// TwinCAT 3 PLC project Carro_Basico_PLC
// ProgramVersion: 3.1.4024.0
// libraries:
//   Tc2_Standard, * (Beckhoff Automation GmbH)
//   Tc2_System, * (Beckhoff Automation GmbH)
//   Tc3_Module, * (Beckhoff Automation GmbH)
//   VisuDialogs, * (System)
// project tree:
//   / GlobalTextList.TcGTLO, PlcTask.TcTTO, Visualization Manager.TcVMO (not stored)
//   POUs/ FB_Blink.TcPOU (not stored), FB_Carro_DRC_LD.TcPOU, FB_Carro_GRF_LD_M.TcPOU (not stored), FB_Carro_GRF_SFC.TcPOU, FB_Carro_GRF_ST.TcPOU, MAIN.TcPOU
//   VISUs/ V_Carro.TcVIS
// real-time tasks:
//   TASK PlcTask: cycle T#10ms, priority 20, ADS port 350

CONFIGURATION Carro_Basico_PLC
    RESOURCE PLC ON TwinCAT3
        TASK PlcTask(INTERVAL := T#10ms, PRIORITY := 20);
        PROGRAM MAIN WITH PlcTask : MAIN;
    END_RESOURCE
END_CONFIGURATION

// ---- POUs/MAIN.TcPOU
PROGRAM MAIN
VAR
    // Carro: FB_Carro_DRC_LD;
    // Carro: FB_Carro_GRF_SFC;
    // Carro: FB_Carro_GRF_ST;
    Carro: FB_Carro_GRF_LD_M;
END_VAR

Carro();

END_PROGRAM

// ---- POUs/FB_Carro_DRC_LD.TcPOU
FUNCTION_BLOCK FB_Carro_DRC_LD
VAR_INPUT
    ManiobrasTotales: UINT := 2;
    TiempoEspera: TIME := T#2S;
END_VAR
VAR_OUTPUT
    ManiobrasPendientes: UINT;
    TiempoPendiente: TIME;
END_VAR
VAR
    // Estados futuros
    MarchaDerechaFuturo: BOOL;
    MarchaIzquierdaFuturo: BOOL;
    
    // Bloques funcionales
    FlancoPulsadorMarcha: R_TRIG;
    Intermitencia: FB_Blink;
    TemporizadorEspera: TON;
    ContadorManiobras: CTD;
    
    // Entradas
    i_PulsadorMarcha AT %I*: BOOL;
    i_FinalCarreraIzquierda AT %I*: BOOL := TRUE;
    i_FinalCarreraDerecha AT %I*: BOOL;
    
    // Salidas
    o_MarchaIzquierda AT %I*: BOOL;
    o_MarchaDerecha AT %I*: BOOL;
    o_LamparaMarcha AT %I*: BOOL;
END_VAR

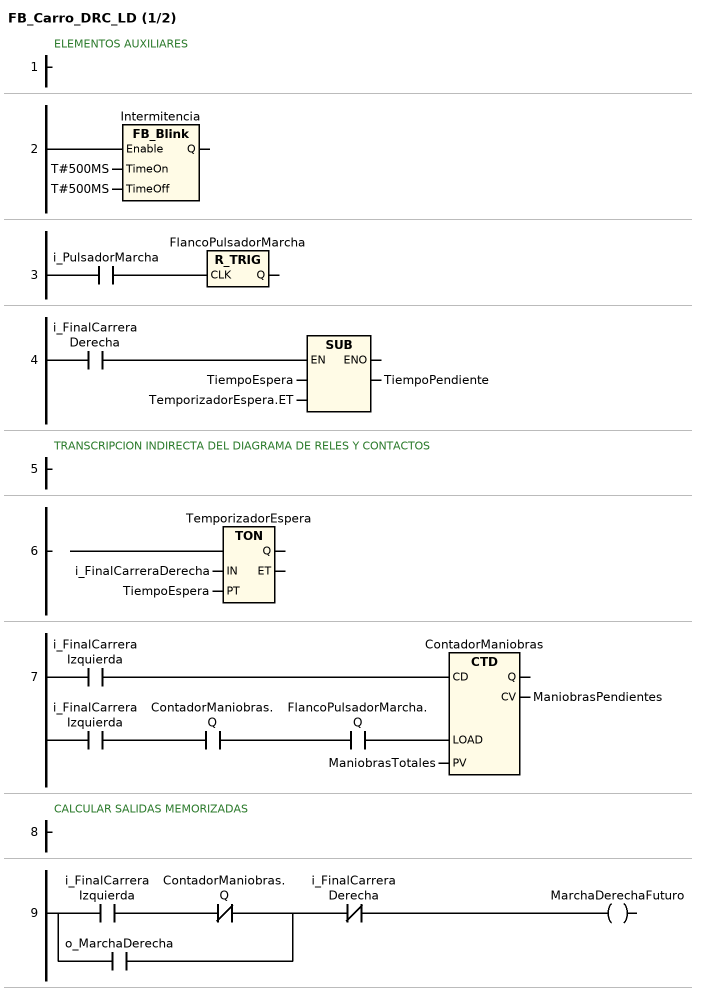
// NETWORK 1
// ELEMENTOS AUXILIARES

// NETWORK 2
Intermitencia(Enable := TRUE, TimeOn := T#500MS, TimeOff := T#500MS); // FB_Blink

// NETWORK 3
FlancoPulsadorMarcha(CLK := i_PulsadorMarcha); // R_TRIG

// NETWORK 4
IF i_FinalCarreraDerecha THEN TiempoPendiente := TiempoEspera - TemporizadorEspera.ET; END_IF

// NETWORK 5
// TRANSCRIPCION INDIRECTA DEL DIAGRAMA DE RELES Y CONTACTOS

// NETWORK 6
TemporizadorEspera(IN := i_FinalCarreraDerecha, PT := TiempoEspera); // TON

// NETWORK 7
ContadorManiobras(
    CD := i_FinalCarreraIzquierda,
    LOAD := i_FinalCarreraIzquierda AND ContadorManiobras.Q AND FlancoPulsadorMarcha.Q,
    PV := ManiobrasTotales,
    CV => ManiobrasPendientes); // CTD

// NETWORK 8
// CALCULAR SALIDAS MEMORIZADAS

// NETWORK 9
MarchaDerechaFuturo := (i_FinalCarreraIzquierda AND NOT ContadorManiobras.Q OR o_MarchaDerecha) AND NOT i_FinalCarreraDerecha;

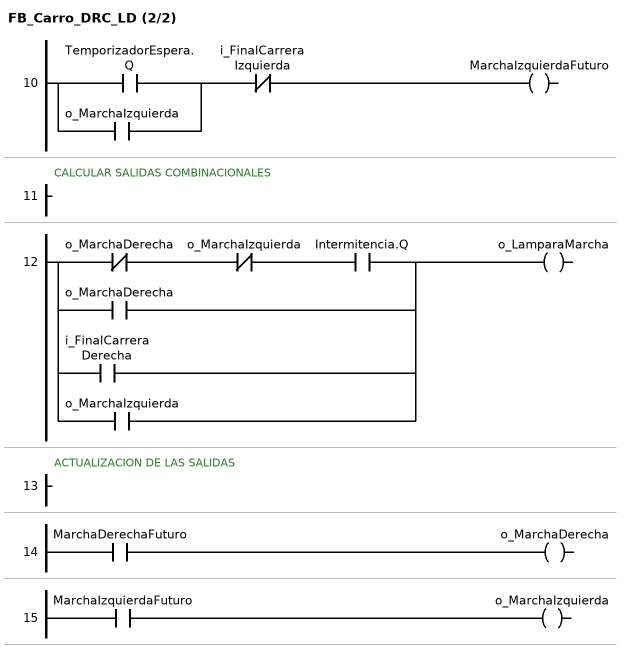
// NETWORK 10
MarchaIzquierdaFuturo := (TemporizadorEspera.Q OR o_MarchaIzquierda) AND NOT i_FinalCarreraIzquierda;

// NETWORK 11
// CALCULAR SALIDAS COMBINACIONALES

// NETWORK 12
o_LamparaMarcha := NOT o_MarchaDerecha AND NOT o_MarchaIzquierda AND Intermitencia.Q OR o_MarchaDerecha OR i_FinalCarreraDerecha OR o_MarchaIzquierda;

// NETWORK 13
// ACTUALIZACION DE LAS SALIDAS

// NETWORK 14
o_MarchaDerecha := MarchaDerechaFuturo;

// NETWORK 15
o_MarchaIzquierda := MarchaIzquierdaFuturo;

END_FUNCTION_BLOCK

// ---- POUs/FB_Carro_GRF_SFC.TcPOU
FUNCTION_BLOCK FB_Carro_GRF_SFC
// Transcripción del grafcet (GRF -> SFC)
VAR_INPUT
    ManiobrasTotales: UINT := 2;
    TiempoEspera: TIME := T#2S;
END_VAR
VAR_OUTPUT
    ManiobrasPendientes: UINT;
    TiempoPendiente: TIME;
END_VAR
VAR
    // Bloques funcionales
    FlancoPulsadorMarcha: R_TRIG;
    Intermitencia: FB_Blink;
    
    // Entradas
    i_PulsadorMarcha AT %I*: BOOL;
    i_FinalCarreraIzquierda AT %I*: BOOL := TRUE;
    i_FinalCarreraDerecha AT %I*: BOOL;
    
    // Salidas
    o_MarchaIzquierda AT %I*: BOOL;
    o_MarchaDerecha AT %I*: BOOL;
    o_LamparaMarcha AT %I*: BOOL;
END_VAR

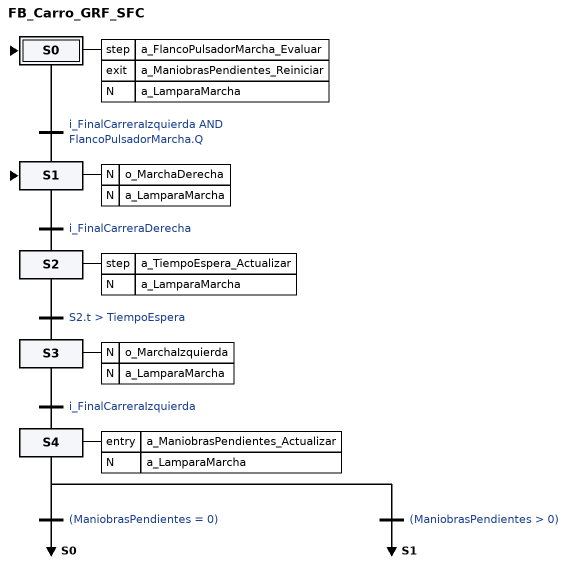
INITIAL_STEP S0:
    a_FlancoPulsadorMarcha_Evaluar(N);  // step action
    a_ManiobrasPendientes_Reiniciar(P0);  // exit action
    a_LamparaMarcha(N);
END_STEP
TRANSITION FROM S0 TO S1
    := i_FinalCarreraIzquierda AND FlancoPulsadorMarcha.Q;
END_TRANSITION
STEP S1:
    o_MarchaDerecha(N);
    a_LamparaMarcha(N);
END_STEP
TRANSITION FROM S1 TO S2
    := i_FinalCarreraDerecha;
END_TRANSITION
STEP S2:
    a_TiempoEspera_Actualizar(N);  // step action
    a_LamparaMarcha(N);
END_STEP
TRANSITION FROM S2 TO S3
    := S2.t > TiempoEspera;
END_TRANSITION
STEP S3:
    o_MarchaIzquierda(N);
    a_LamparaMarcha(N);
END_STEP
TRANSITION FROM S3 TO S4
    := i_FinalCarreraIzquierda;
END_TRANSITION
STEP S4:
    a_ManiobrasPendientes_Actualizar(P1);  // entry action
    a_LamparaMarcha(N);
END_STEP
TRANSITION FROM S4 TO S0
    := (ManiobrasPendientes = 0);
END_TRANSITION
TRANSITION FROM S4 TO S1
    := (ManiobrasPendientes > 0);
END_TRANSITION

ACTION a_FlancoPulsadorMarcha_Evaluar:
FlancoPulsadorMarcha(CLK := i_PulsadorMarcha);
END_ACTION

ACTION a_LamparaMarcha:
Intermitencia();

o_LamparaMarcha := (S0.x AND Intermitencia.Q) OR S1.x OR S2.x OR S3.x OR S4.x;
END_ACTION

ACTION a_ManiobrasPendientes_Actualizar:
IF (ManiobrasPendientes > 0) THEN
    ManiobrasPendientes := ManiobrasPendientes - 1;
END_IF;
END_ACTION

ACTION a_ManiobrasPendientes_Reiniciar:
ManiobrasPendientes := ManiobrasTotales;
END_ACTION

ACTION a_TiempoEspera_Actualizar:
IF TiempoEspera >= S2.t THEN
    TiempoPendiente := TiempoEspera - S2.t;
END_IF;
END_ACTION

END_FUNCTION_BLOCK

// ---- POUs/FB_Carro_GRF_ST.TcPOU
FUNCTION_BLOCK FB_Carro_GRF_ST
// Transcripción del grafcet (GRF -> ST)
VAR_INPUT
    ManiobrasTotales: UINT := 2;
    TiempoEspera: TIME := T#2S;
END_VAR
VAR_OUTPUT
    ManiobrasPendientes: UINT;
    TiempoPendiente: TIME;
END_VAR
VAR
    Estado: (E_REPOSO, E_DERECHA, E_ESPERA, E_IZQUIERDA, E_FIN);
    
    // Bloques funcionales
    FlancoPulsadorMarcha: R_TRIG;
    Intermitencia: FB_Blink;
    TemporizadorEspera: TON;
    
    // Entradas
    i_PulsadorMarcha AT %I*: BOOL;
    i_FinalCarreraIzquierda AT %I*: BOOL := TRUE;
    i_FinalCarreraDerecha AT %I*: BOOL;
    
    // Salidas
    o_MarchaIzquierda AT %I*: BOOL;
    o_MarchaDerecha AT %I*: BOOL;
    o_LamparaMarcha AT %I*: BOOL;
END_VAR

// BLOQUES FUNCIONALES
Intermitencia(Enable := (Estado = E_REPOSO));
TemporizadorEspera(IN := (Estado = E_ESPERA), PT := TiempoEspera);

// FUNCION DE ESTADO
CASE Estado OF
    E_REPOSO:
        // Acción principal
        FlancoPulsadorMarcha(CLK := i_PulsadorMarcha);
        
        IF i_FinalCarreraIzquierda AND FlancoPulsadorMarcha.Q THEN
            // Acción de salida
            ManiobrasPendientes := ManiobrasTotales;
            
            Estado := E_DERECHA;
		END_IF;
    E_DERECHA:
        IF i_FinalCarreraDerecha THEN            
            Estado := E_ESPERA;
		END_IF;
    E_ESPERA:
        // Acción principal
        IF (TiempoEspera >= TemporizadorEspera.ET) THEN
            TiempoPendiente := TiempoEspera - TemporizadorEspera.ET;
        END_IF;

        IF TemporizadorEspera.Q  THEN
            Estado := E_IZQUIERDA;
		END_IF;
    E_IZQUIERDA:
        IF i_FinalCarreraIzquierda THEN
            // Acción de entrada del siguiente estado
            IF (ManiobrasPendientes > 0) THEN 
                ManiobrasPendientes := ManiobrasPendientes - 1;
            END_IF;
                
            Estado := E_FIN;
		END_IF;
    E_FIN:
        IF (ManiobrasPendientes = 0) THEN
            Estado := E_REPOSO;
        ELSIF (ManiobrasPendientes > 0) THEN
            Estado := E_DERECHA;
		END_IF;
END_CASE;

// FUNCION DE SALIDA
o_MarchaDerecha := (Estado = E_DERECHA);
o_MarchaIzquierda := (Estado = E_IZQUIERDA);
o_LamparaMarcha := (Estado <> E_REPOSO) OR Intermitencia.Q;

END_FUNCTION_BLOCK

// ---- GlobalTextList.TcGTLO
TEXTLIST GlobalTextList
  831 = '%d'
  250 = '%t[ss.ms] s'
  827 = '3'
  39 = '4'
  774 = '7'
  772 = '8'
  311 = 'Carro'
  703 = 'CARRO BÁSICO'
  744 = 'Dch'
  522 = 'Espera'
  24 = 'Izq'
  314 = 'Maniobras'
  92 = 'Marcha'
  773 = 'Marcha derecha'
  909 = 'Panel'
  273 = 'Pendiente'
  53 = 'Pendientes'
  449 = 'Tiempos'
  498 = 'Totales'
END_TEXTLIST

// ---- VISUs/V_Carro.TcVIS
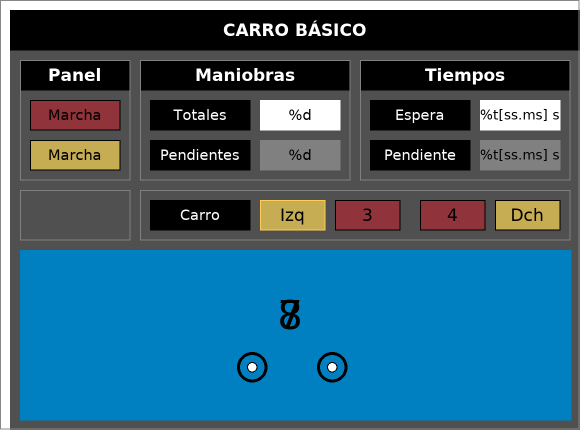
VISUALIZATION V_Carro  // 580x430
    Rectangle (10,50 570x380)
    Rectangle (140,190 430x50)
    Rectangle (20,60 110x30), "Panel"
    Rectangle (20,60 110x120)
    Rectangle (360,60 210x30), "Tiempos"
    Rectangle (360,60 210x120)
    Rectangle (10,10 570x40), "CARRO BÁSICO"
    RoundedRectangle (370,100 100x30), "Espera"
    Rectangle (140,60 210x30), "Maniobras"
    Rectangle (480,100 80x30), "%t[ss.ms] s", text variable: MAIN.Carro.TiempoEspera
        OnMouseClick: write the text variable via Default
    RoundedRectangle (370,140 100x30), "Pendiente"
    Rectangle (480,140 80x30), "%t[ss.ms] s", text variable: MAIN.Carro.TiempoPendiente
        OnMouseClick: write the text variable via Default
    Rectangle (30,100 90x30), "Marcha", colour toggle: MAIN.Carro.o_LamparaMarcha
        tap MAIN.Carro.o_LamparaMarcha
    Rectangle (30,140 90x30), "Marcha", colour toggle: MAIN.Carro.i_PulsadorMarcha
        toggle MAIN.Carro.i_PulsadorMarcha
    Rectangle (140,60 210x120)
    RoundedRectangle (150,100 100x30), "Totales"
    Rectangle (260,100 80x30), "%d", text variable: MAIN.Carro.ManiobrasTotales
        OnMouseClick: write the text variable via Default
    RoundedRectangle (150,140 100x30), "Pendientes"
    Rectangle (260,140 80x30), "%d", text variable: MAIN.Carro.ManiobrasPendientes
        OnMouseClick: write the text variable via Default
    Rectangle (20,250 551x170)
    Polyline (477,390)
    Polygon (105,385), colour toggle: MAIN.Carro.i_FinalCarreraIzquierda
        p2738717112: SEL (MAIN.Carro.i_FinalCarreraIzquierda, 0, 5)
        toggle MAIN.Carro.i_FinalCarreraIzquierda
    Polygon (435,385), colour toggle: MAIN.Carro.i_FinalCarreraDerecha
        p2738717112: SEL (MAIN.Carro.i_FinalCarreraDerecha, 0, 5)
        toggle MAIN.Carro.i_FinalCarreraDerecha
    Group (211,281 158x98), invisible if: MAIN.Carro.i_FinalCarreraIzquierda AND MAIN.Carro.i_FinalCarreraDerecha
        p3560616238: SEL (MAIN.Carro.i_FinalCarreraDerecha, SEL (MAIN.Carro.i_FinalCarreraIzquierda, 0, -125), 125)
        Polygon (0,0)
        Polygon (115,80)
        Group (106,71 28x28)
            Ellipse (0,0 30x30)
            Ellipse (10,10 10x10)
        Polygon (35,80)
        Group (26,71 28x28)
            Ellipse (0,0 30x30)
            Ellipse (10,10 10x10)
    Rectangle (270,295 40x40), "8", tooltip "Marcha derecha", invisible if: NOT MAIN.Carro.o_MarchaDerecha
        p3560616238: SEL (MAIN.Carro.i_FinalCarreraDerecha, SEL (MAIN.Carro.i_FinalCarreraIzquierda, 0, -125), 125)
    Rectangle (270,295 40x40), "7", invisible if: NOT MAIN.Carro.o_MarchaIzquierda
        p3560616238: SEL (MAIN.Carro.i_FinalCarreraDerecha, SEL (MAIN.Carro.i_FinalCarreraIzquierda, 0, -125), 125)
    RoundedRectangle (150,200 100x30), "Carro"
    Rectangle (335,200 65x30), "3", colour toggle: MAIN.Carro.o_MarchaIzquierda
        toggle MAIN.Carro.o_MarchaIzquierda
    Rectangle (420,200 65x30), "4", colour toggle: MAIN.Carro.o_MarchaDerecha
        toggle MAIN.Carro.o_MarchaDerecha
    Rectangle (260,200 65x30), "Izq", colour toggle: MAIN.Carro.i_FinalCarreraIzquierda
        toggle MAIN.Carro.i_FinalCarreraIzquierda
    Rectangle (495,200 65x30), "Dch", colour toggle: MAIN.Carro.i_FinalCarreraDerecha
        toggle MAIN.Carro.i_FinalCarreraDerecha
    Rectangle (20,190 110x50)
END_VISUALIZATION
